PROGRAM ST3_ETANCHEITE
VAR
	STEP: INT := 0;
	JIG_STATUS_R_TRIG: R_TRIG;
	START_TAMPO_MISE_SOUS_PRESSION: BOOL;
	TAMPO_MISE_SOUS_PRESSION: TON;
	START_TAMPO_STABILISATION: BOOL;
	TAMPO_STABILISATION: TON;
	START_TAMPO_MESURE: BOOL;
	TAMPO_MESURE: TON;
	PRESSION_DEBUT: REAL;
	PRESSION_FIN: REAL;
END_VAR

(*******************************************************
*
* Station 3 - Etanchéité
*
*
*********************************************************)
IF NOT(GEMMA.STEP='F1') THEN
	STEP:=0;
END_IF;


CASE STEP OF

0: (*Init*)

	ST3_3V4 := FALSE;
	ST3_3V5 := FALSE;
	ST3_3V10 := FALSE;
	ST3_3V11 := FALSE;
	ST3_3V12 := FALSE;
	
	FLAGS.ST3_RELEASE_CARRIER := FALSE;
	
	START_TAMPO_MISE_SOUS_PRESSION := FALSE;
	START_TAMPO_STABILISATION := FALSE;
	START_TAMPO_MESURE := FALSE;

	
	STEP := STEP + 10;
	
10: (*Attend une palette / flanc montant du status*)

	IF JIG_STATUS_R_TRIG.Q THEN
		STEP := STEP + 10;
	END_IF;
	
20: (*Descend le vérin du dessus*)

	ST3_3V4 := TRUE;
	STEP := STEP + 10;
	
30: (*Attend vérin dessus sorti*)

	IF ST3_3B4 THEN
		STEP := STEP + 10;
	END_IF;

40: (*Monte le vérin du dessous*)

	ST3_3V5 := TRUE;
	STEP := STEP + 10;
	
50: (*Attend vérin dessus sorti*)

	IF ST3_3B5 THEN
		STEP := 100;
	END_IF;
	
	
(**************************************************************************)
100: (*Mise sous pression de la cartouche*)

	ST3_3V10 := TRUE;
	ST3_3V11 := FALSE;
	ST3_3V12 := TRUE;
	
	START_TAMPO_MISE_SOUS_PRESSION := TRUE;
	
	STEP := STEP + 10;
	
	
110: (*Tampo pour la mise sous pression de la cartouche*)

	IF TAMPO_MISE_SOUS_PRESSION.Q THEN
		START_TAMPO_MISE_SOUS_PRESSION := FALSE;
		STEP := STEP + 10;
	END_IF;

120: (*Start stabilisation*)

	START_TAMPO_STABILISATION := TRUE;
	ST3_3V10 := FALSE;
	
	STEP := STEP + 10;	

130: (*Tampo pour la stabilisation de la pression dans la cartouche*)

	IF TAMPO_STABILISATION.Q THEN
		START_TAMPO_STABILISATION := FALSE;
		STEP := STEP + 10;
	END_IF;
	
140: (*Start stabilisation*)

	START_TAMPO_MESURE := TRUE;
	ST3_3V12 := FALSE;
	PRESSION_DEBUT := 0; (* Mesure de la pression au début du test *)
	
	STEP := STEP + 10;	

150: (*Tampo pour la stabilisation de la pression dans la cartouche*)

	IF TAMPO_MESURE.Q THEN
		START_TAMPO_MESURE := FALSE;
		PRESSION_FIN := 0; (* Mesure de la pression à la fin du test *)
		ST3_DELTA_P := PRESSION_FIN - PRESSION_DEBUT; (* Calcule de la chutte de pression *)
		STEP := STEP + 10;
	END_IF;
	
160: (*Fin mesure, dépressiorisation de la cartouche*)

	ST3_3V10 := FALSE;
	ST3_3V11 := TRUE;
	ST3_3V12 := TRUE;
	
	STEP := 300;	
	
	

(**************************************************************************)	

300: (*Descend le vérin du dessous*)

	ST3_3V5 := FALSE;
	STEP := STEP + 10;
	
310: (*Monte le vérin du dessus*)

	ST3_3V4 := FALSE;
	STEP := STEP + 10;

320: (*Libère la palette*)

	FLAGS.ST3_RELEASE_CARRIER := TRUE;
	STEP := 0;


ELSE
    (*default case*);
END_CASE;

(*FBs*)

TAMPO_MISE_SOUS_PRESSION(IN:= START_TAMPO_MISE_SOUS_PRESSION, PT:= PUMP_PARAMS.ST3_TEMPS_MISE_SOUS_PRESSION);
TAMPO_STABILISATION(IN:= START_TAMPO_STABILISATION, PT:= PUMP_PARAMS.ST3_TEMPS_STABILISATION);
TAMPO_MESURE(IN:= START_TAMPO_MESURE, PT:= PUMP_PARAMS.ST3_TEMPS_MESURE);
JIG_STATUS_R_TRIG(CLK:= CONVEYOR.JIG_ST3.STATUS);
PROG_STEPS.ST3:=STEP;

END_PROGRAM

(* stored: Version 1.1.0.1, ProductVersion 3.1.0.26
   POU ST3_ETANCHEITE: Id {4c8d0ed2-e515-4489-ae28-5ece9354e79b} *)
